Staubli VAL3: TRAJ.dtx

public Traies tTraj{}
